// TIA Portal V19 export
FUNCTION "AI SCALING" : Void   // FC5, LAD
{ S7_Optimized_Access := 'TRUE' }
// stored: SetENOAutomatically false
BEGIN

REGION Network 1: OXIDATION REDUCTION POTENTIO METER 301
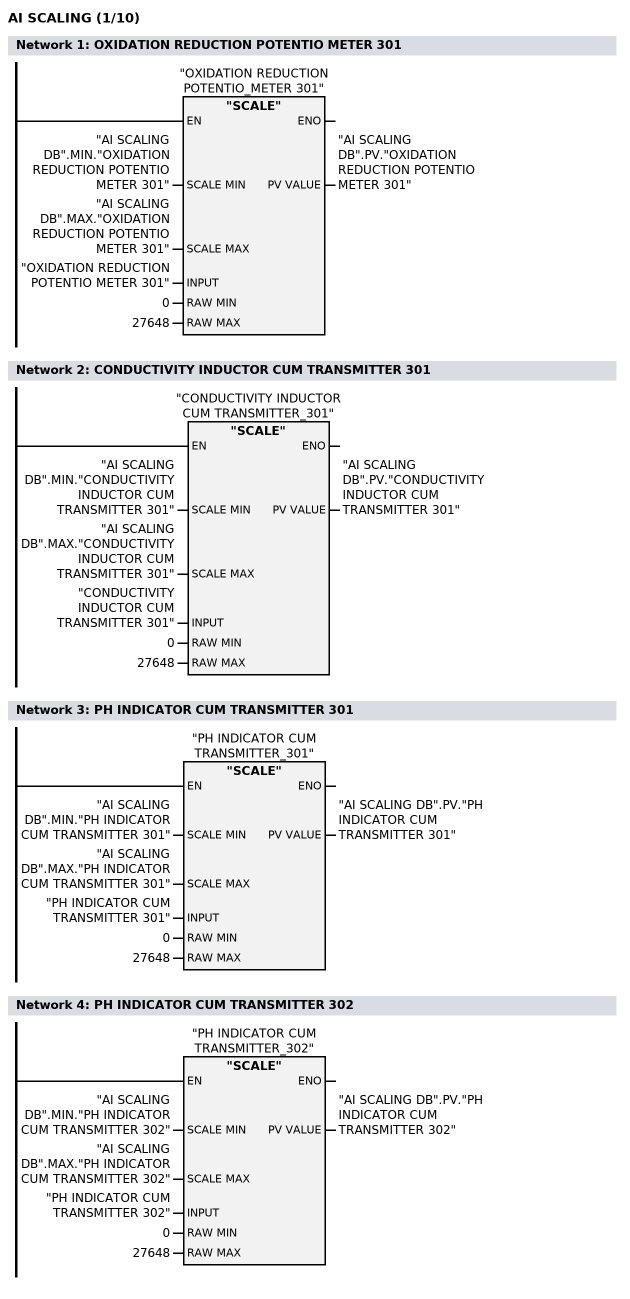
   RUNG wire#powerrail
      "OXIDATION REDUCTION POTENTIO_METER 301"("SCALE MIN" := "AI SCALING DB".MIN."OXIDATION REDUCTION POTENTIO METER 301", "SCALE MAX" := "AI SCALING DB".MAX."OXIDATION REDUCTION POTENTIO METER 301", INPUT := "OXIDATION REDUCTION POTENTIO METER 301", "RAW MIN" := 0, "RAW MAX" := 27648, "PV VALUE" => "AI SCALING DB".PV."OXIDATION REDUCTION POTENTIO METER 301")
   END_RUNG
   // the same network as SCL:
   "OXIDATION REDUCTION POTENTIO_METER 301"("SCALE MIN" := "AI SCALING DB".MIN."OXIDATION REDUCTION POTENTIO METER 301",   // "SCALE"
                           "SCALE MAX" := "AI SCALING DB".MAX."OXIDATION REDUCTION POTENTIO METER 301",
                           INPUT := "OXIDATION REDUCTION POTENTIO METER 301",
                           "RAW MIN" := 0,
                           "RAW MAX" := 27648,
                           "PV VALUE" => "AI SCALING DB".PV."OXIDATION REDUCTION POTENTIO METER 301");
END_REGION

REGION Network 2: CONDUCTIVITY INDUCTOR CUM TRANSMITTER 301
   RUNG wire#powerrail
      "CONDUCTIVITY INDUCTOR CUM TRANSMITTER_301"("SCALE MIN" := "AI SCALING DB".MIN."CONDUCTIVITY INDUCTOR CUM TRANSMITTER 301", "SCALE MAX" := "AI SCALING DB".MAX."CONDUCTIVITY INDUCTOR CUM TRANSMITTER 301", INPUT := "CONDUCTIVITY INDUCTOR CUM TRANSMITTER 301", "RAW MIN" := 0, "RAW MAX" := 27648, "PV VALUE" => "AI SCALING DB".PV."CONDUCTIVITY INDUCTOR CUM TRANSMITTER 301")
   END_RUNG
   // the same network as SCL:
   "CONDUCTIVITY INDUCTOR CUM TRANSMITTER_301"("SCALE MIN" := "AI SCALING DB".MIN."CONDUCTIVITY INDUCTOR CUM TRANSMITTER 301",   // "SCALE"
                           "SCALE MAX" := "AI SCALING DB".MAX."CONDUCTIVITY INDUCTOR CUM TRANSMITTER 301",
                           INPUT := "CONDUCTIVITY INDUCTOR CUM TRANSMITTER 301",
                           "RAW MIN" := 0,
                           "RAW MAX" := 27648,
                           "PV VALUE" => "AI SCALING DB".PV."CONDUCTIVITY INDUCTOR CUM TRANSMITTER 301");
END_REGION

REGION Network 3: PH INDICATOR CUM TRANSMITTER 301
   RUNG wire#powerrail
      "PH INDICATOR CUM TRANSMITTER_301"("SCALE MIN" := "AI SCALING DB".MIN."PH INDICATOR CUM TRANSMITTER 301", "SCALE MAX" := "AI SCALING DB".MAX."PH INDICATOR CUM TRANSMITTER 301", INPUT := "PH INDICATOR CUM TRANSMITTER 301", "RAW MIN" := 0, "RAW MAX" := 27648, "PV VALUE" => "AI SCALING DB".PV."PH INDICATOR CUM TRANSMITTER 301")
   END_RUNG
   // the same network as SCL:
   "PH INDICATOR CUM TRANSMITTER_301"("SCALE MIN" := "AI SCALING DB".MIN."PH INDICATOR CUM TRANSMITTER 301",   // "SCALE"
                           "SCALE MAX" := "AI SCALING DB".MAX."PH INDICATOR CUM TRANSMITTER 301",
                           INPUT := "PH INDICATOR CUM TRANSMITTER 301",
                           "RAW MIN" := 0,
                           "RAW MAX" := 27648,
                           "PV VALUE" => "AI SCALING DB".PV."PH INDICATOR CUM TRANSMITTER 301");
END_REGION

REGION Network 4: PH INDICATOR CUM TRANSMITTER 302
   RUNG wire#powerrail
      "PH INDICATOR CUM TRANSMITTER_302"("SCALE MIN" := "AI SCALING DB".MIN."PH INDICATOR CUM TRANSMITTER 302", "SCALE MAX" := "AI SCALING DB".MAX."PH INDICATOR CUM TRANSMITTER 302", INPUT := "PH INDICATOR CUM TRANSMITTER 302", "RAW MIN" := 0, "RAW MAX" := 27648, "PV VALUE" => "AI SCALING DB".PV."PH INDICATOR CUM TRANSMITTER 302")
   END_RUNG
   // the same network as SCL:
   "PH INDICATOR CUM TRANSMITTER_302"("SCALE MIN" := "AI SCALING DB".MIN."PH INDICATOR CUM TRANSMITTER 302",   // "SCALE"
                           "SCALE MAX" := "AI SCALING DB".MAX."PH INDICATOR CUM TRANSMITTER 302",
                           INPUT := "PH INDICATOR CUM TRANSMITTER 302",
                           "RAW MIN" := 0,
                           "RAW MAX" := 27648,
                           "PV VALUE" => "AI SCALING DB".PV."PH INDICATOR CUM TRANSMITTER 302");
END_REGION

REGION Network 5: CONDUCTIVITY INDICATOR CUM TRANSMITTER 302
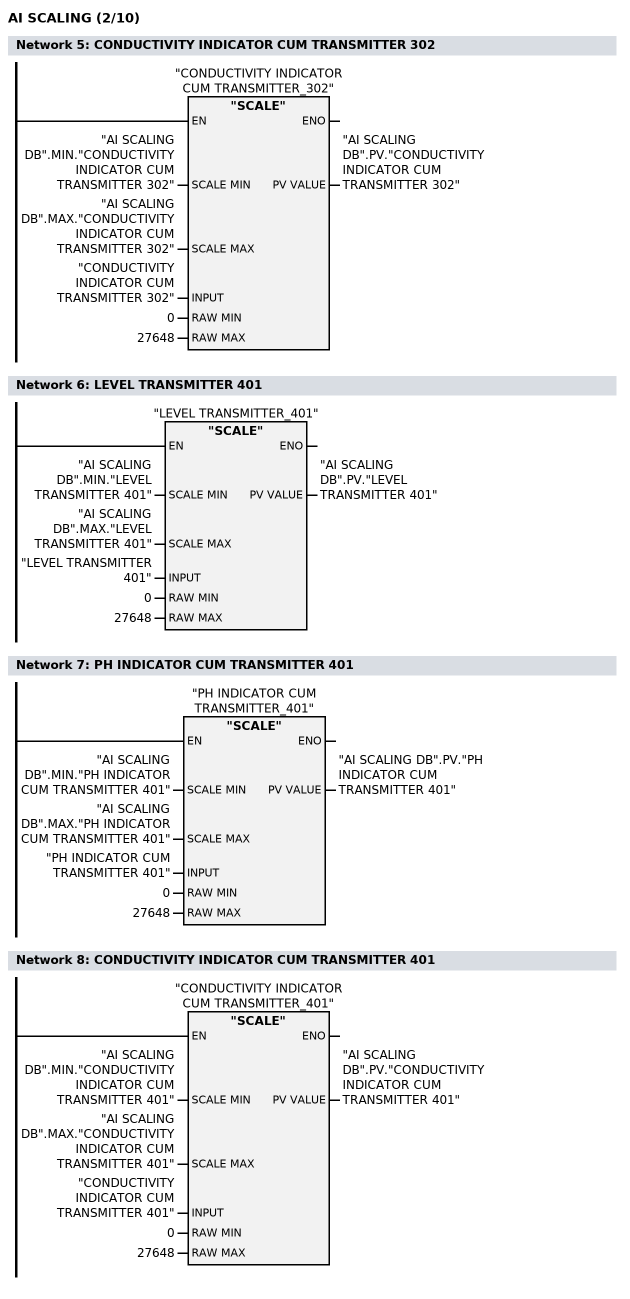
   RUNG wire#powerrail
      "CONDUCTIVITY INDICATOR CUM TRANSMITTER_302"("SCALE MIN" := "AI SCALING DB".MIN."CONDUCTIVITY INDICATOR CUM TRANSMITTER 302", "SCALE MAX" := "AI SCALING DB".MAX."CONDUCTIVITY INDICATOR CUM TRANSMITTER 302", INPUT := "CONDUCTIVITY INDICATOR CUM TRANSMITTER 302", "RAW MIN" := 0, "RAW MAX" := 27648, "PV VALUE" => "AI SCALING DB".PV."CONDUCTIVITY INDICATOR CUM TRANSMITTER 302")
   END_RUNG
   // the same network as SCL:
   "CONDUCTIVITY INDICATOR CUM TRANSMITTER_302"("SCALE MIN" := "AI SCALING DB".MIN."CONDUCTIVITY INDICATOR CUM TRANSMITTER 302",   // "SCALE"
                           "SCALE MAX" := "AI SCALING DB".MAX."CONDUCTIVITY INDICATOR CUM TRANSMITTER 302",
                           INPUT := "CONDUCTIVITY INDICATOR CUM TRANSMITTER 302",
                           "RAW MIN" := 0,
                           "RAW MAX" := 27648,
                           "PV VALUE" => "AI SCALING DB".PV."CONDUCTIVITY INDICATOR CUM TRANSMITTER 302");
END_REGION

REGION Network 6: LEVEL TRANSMITTER 401
   RUNG wire#powerrail
      "LEVEL TRANSMITTER_401"("SCALE MIN" := "AI SCALING DB".MIN."LEVEL TRANSMITTER 401", "SCALE MAX" := "AI SCALING DB".MAX."LEVEL TRANSMITTER 401", INPUT := "LEVEL TRANSMITTER 401", "RAW MIN" := 0, "RAW MAX" := 27648, "PV VALUE" => "AI SCALING DB".PV."LEVEL TRANSMITTER 401")
   END_RUNG
   // the same network as SCL:
   "LEVEL TRANSMITTER_401"("SCALE MIN" := "AI SCALING DB".MIN."LEVEL TRANSMITTER 401",   // "SCALE"
                           "SCALE MAX" := "AI SCALING DB".MAX."LEVEL TRANSMITTER 401",
                           INPUT := "LEVEL TRANSMITTER 401",
                           "RAW MIN" := 0,
                           "RAW MAX" := 27648,
                           "PV VALUE" => "AI SCALING DB".PV."LEVEL TRANSMITTER 401");
END_REGION

REGION Network 7: PH INDICATOR CUM TRANSMITTER 401
   RUNG wire#powerrail
      "PH INDICATOR CUM TRANSMITTER_401"("SCALE MIN" := "AI SCALING DB".MIN."PH INDICATOR CUM TRANSMITTER 401", "SCALE MAX" := "AI SCALING DB".MAX."PH INDICATOR CUM TRANSMITTER 401", INPUT := "PH INDICATOR CUM TRANSMITTER 401", "RAW MIN" := 0, "RAW MAX" := 27648, "PV VALUE" => "AI SCALING DB".PV."PH INDICATOR CUM TRANSMITTER 401")
   END_RUNG
   // the same network as SCL:
   "PH INDICATOR CUM TRANSMITTER_401"("SCALE MIN" := "AI SCALING DB".MIN."PH INDICATOR CUM TRANSMITTER 401",   // "SCALE"
                           "SCALE MAX" := "AI SCALING DB".MAX."PH INDICATOR CUM TRANSMITTER 401",
                           INPUT := "PH INDICATOR CUM TRANSMITTER 401",
                           "RAW MIN" := 0,
                           "RAW MAX" := 27648,
                           "PV VALUE" => "AI SCALING DB".PV."PH INDICATOR CUM TRANSMITTER 401");
END_REGION

REGION Network 8: CONDUCTIVITY INDICATOR CUM TRANSMITTER 401
   RUNG wire#powerrail
      "CONDUCTIVITY INDICATOR CUM TRANSMITTER_401"("SCALE MIN" := "AI SCALING DB".MIN."CONDUCTIVITY INDICATOR CUM TRANSMITTER 401", "SCALE MAX" := "AI SCALING DB".MAX."CONDUCTIVITY INDICATOR CUM TRANSMITTER 401", INPUT := "CONDUCTIVITY INDICATOR CUM TRANSMITTER 401", "RAW MIN" := 0, "RAW MAX" := 27648, "PV VALUE" => "AI SCALING DB".PV."CONDUCTIVITY INDICATOR CUM TRANSMITTER 401")
   END_RUNG
   // the same network as SCL:
   "CONDUCTIVITY INDICATOR CUM TRANSMITTER_401"("SCALE MIN" := "AI SCALING DB".MIN."CONDUCTIVITY INDICATOR CUM TRANSMITTER 401",   // "SCALE"
                           "SCALE MAX" := "AI SCALING DB".MAX."CONDUCTIVITY INDICATOR CUM TRANSMITTER 401",
                           INPUT := "CONDUCTIVITY INDICATOR CUM TRANSMITTER 401",
                           "RAW MIN" := 0,
                           "RAW MAX" := 27648,
                           "PV VALUE" => "AI SCALING DB".PV."CONDUCTIVITY INDICATOR CUM TRANSMITTER 401");
END_REGION

REGION Network 9: CONFUCTIVITY INDICATOR CUM TRANSMITTER 402
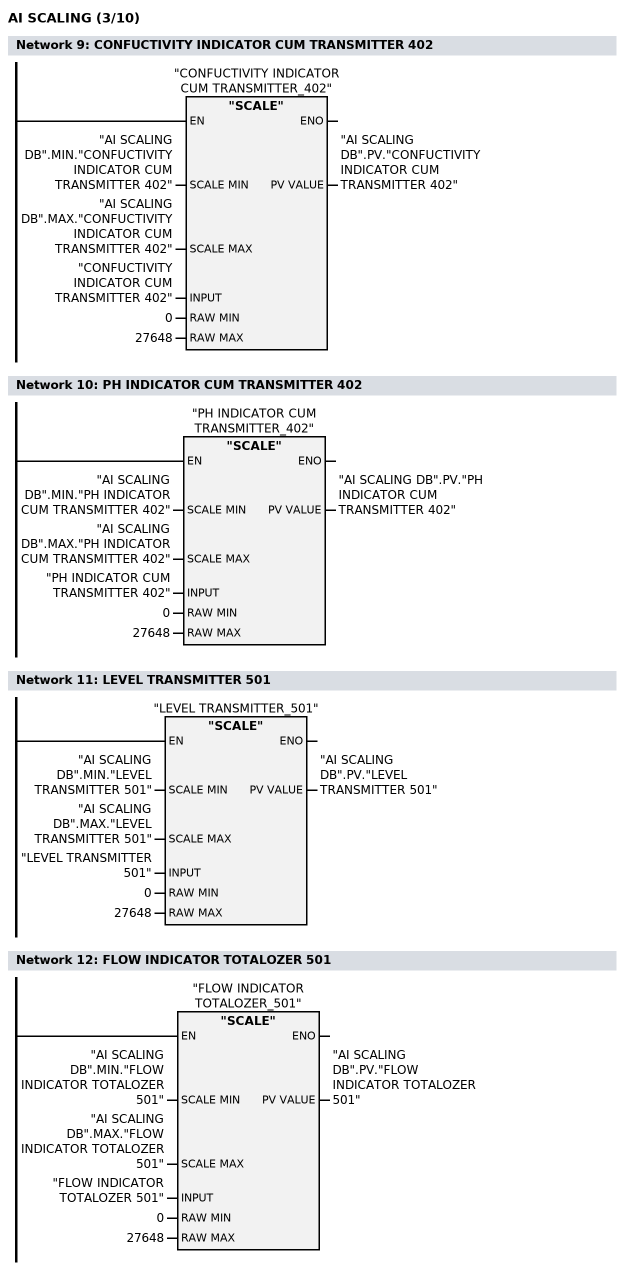
   RUNG wire#powerrail
      "CONFUCTIVITY INDICATOR CUM TRANSMITTER_402"("SCALE MIN" := "AI SCALING DB".MIN."CONFUCTIVITY INDICATOR CUM TRANSMITTER 402", "SCALE MAX" := "AI SCALING DB".MAX."CONFUCTIVITY INDICATOR CUM TRANSMITTER 402", INPUT := "CONFUCTIVITY INDICATOR CUM TRANSMITTER 402", "RAW MIN" := 0, "RAW MAX" := 27648, "PV VALUE" => "AI SCALING DB".PV."CONFUCTIVITY INDICATOR CUM TRANSMITTER 402")
   END_RUNG
   // the same network as SCL:
   "CONFUCTIVITY INDICATOR CUM TRANSMITTER_402"("SCALE MIN" := "AI SCALING DB".MIN."CONFUCTIVITY INDICATOR CUM TRANSMITTER 402",   // "SCALE"
                           "SCALE MAX" := "AI SCALING DB".MAX."CONFUCTIVITY INDICATOR CUM TRANSMITTER 402",
                           INPUT := "CONFUCTIVITY INDICATOR CUM TRANSMITTER 402",
                           "RAW MIN" := 0,
                           "RAW MAX" := 27648,
                           "PV VALUE" => "AI SCALING DB".PV."CONFUCTIVITY INDICATOR CUM TRANSMITTER 402");
END_REGION

REGION Network 10: PH INDICATOR CUM TRANSMITTER 402
   RUNG wire#powerrail
      "PH INDICATOR CUM TRANSMITTER_402"("SCALE MIN" := "AI SCALING DB".MIN."PH INDICATOR CUM TRANSMITTER 402", "SCALE MAX" := "AI SCALING DB".MAX."PH INDICATOR CUM TRANSMITTER 402", INPUT := "PH INDICATOR CUM TRANSMITTER 402", "RAW MIN" := 0, "RAW MAX" := 27648, "PV VALUE" => "AI SCALING DB".PV."PH INDICATOR CUM TRANSMITTER 402")
   END_RUNG
   // the same network as SCL:
   "PH INDICATOR CUM TRANSMITTER_402"("SCALE MIN" := "AI SCALING DB".MIN."PH INDICATOR CUM TRANSMITTER 402",   // "SCALE"
                           "SCALE MAX" := "AI SCALING DB".MAX."PH INDICATOR CUM TRANSMITTER 402",
                           INPUT := "PH INDICATOR CUM TRANSMITTER 402",
                           "RAW MIN" := 0,
                           "RAW MAX" := 27648,
                           "PV VALUE" => "AI SCALING DB".PV."PH INDICATOR CUM TRANSMITTER 402");
END_REGION

REGION Network 11: LEVEL TRANSMITTER 501
   RUNG wire#powerrail
      "LEVEL TRANSMITTER_501"("SCALE MIN" := "AI SCALING DB".MIN."LEVEL TRANSMITTER 501", "SCALE MAX" := "AI SCALING DB".MAX."LEVEL TRANSMITTER 501", INPUT := "LEVEL TRANSMITTER 501", "RAW MIN" := 0, "RAW MAX" := 27648, "PV VALUE" => "AI SCALING DB".PV."LEVEL TRANSMITTER 501")
   END_RUNG
   // the same network as SCL:
   "LEVEL TRANSMITTER_501"("SCALE MIN" := "AI SCALING DB".MIN."LEVEL TRANSMITTER 501",   // "SCALE"
                           "SCALE MAX" := "AI SCALING DB".MAX."LEVEL TRANSMITTER 501",
                           INPUT := "LEVEL TRANSMITTER 501",
                           "RAW MIN" := 0,
                           "RAW MAX" := 27648,
                           "PV VALUE" => "AI SCALING DB".PV."LEVEL TRANSMITTER 501");
END_REGION

REGION Network 12: FLOW INDICATOR TOTALOZER 501
   RUNG wire#powerrail
      "FLOW INDICATOR TOTALOZER_501"("SCALE MIN" := "AI SCALING DB".MIN."FLOW INDICATOR TOTALOZER 501", "SCALE MAX" := "AI SCALING DB".MAX."FLOW INDICATOR TOTALOZER 501", INPUT := "FLOW INDICATOR TOTALOZER 501", "RAW MIN" := 0, "RAW MAX" := 27648, "PV VALUE" => "AI SCALING DB".PV."FLOW INDICATOR TOTALOZER 501")
   END_RUNG
   // the same network as SCL:
   "FLOW INDICATOR TOTALOZER_501"("SCALE MIN" := "AI SCALING DB".MIN."FLOW INDICATOR TOTALOZER 501",   // "SCALE"
                           "SCALE MAX" := "AI SCALING DB".MAX."FLOW INDICATOR TOTALOZER 501",
                           INPUT := "FLOW INDICATOR TOTALOZER 501",
                           "RAW MIN" := 0,
                           "RAW MAX" := 27648,
                           "PV VALUE" => "AI SCALING DB".PV."FLOW INDICATOR TOTALOZER 501");
END_REGION

REGION Network 13: PRESSURE TRANSMITTER 501
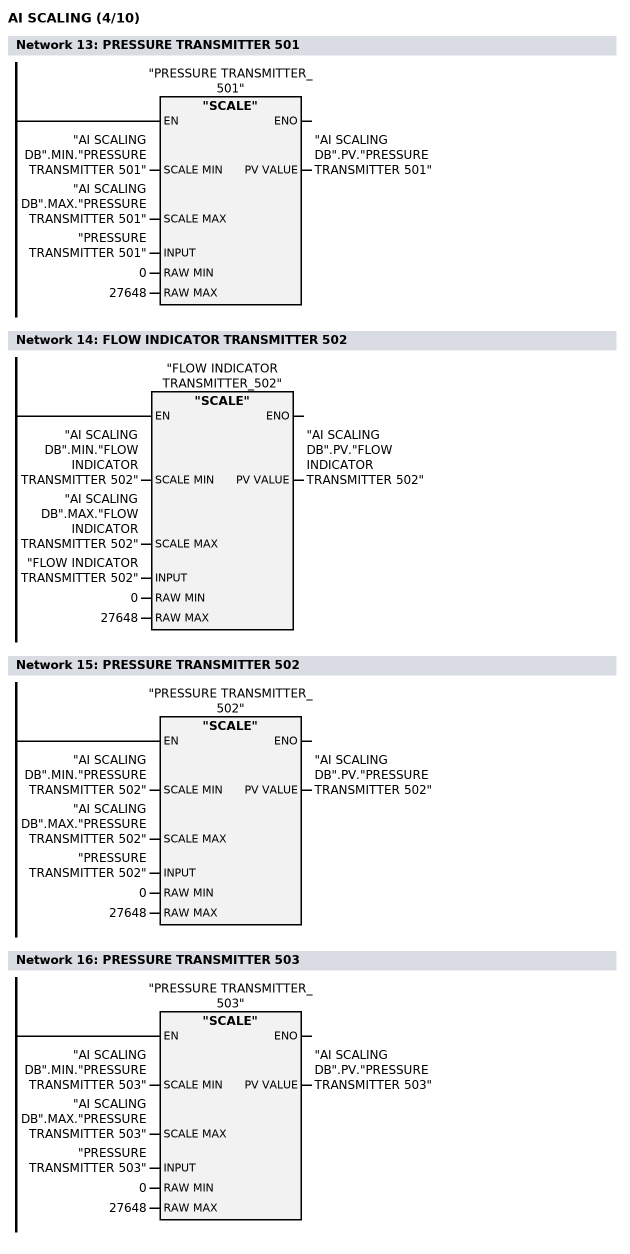
   RUNG wire#powerrail
      "PRESSURE TRANSMITTER_501"("SCALE MIN" := "AI SCALING DB".MIN."PRESSURE TRANSMITTER 501", "SCALE MAX" := "AI SCALING DB".MAX."PRESSURE TRANSMITTER 501", INPUT := "PRESSURE TRANSMITTER 501", "RAW MIN" := 0, "RAW MAX" := 27648, "PV VALUE" => "AI SCALING DB".PV."PRESSURE TRANSMITTER 501")
   END_RUNG
   // the same network as SCL:
   "PRESSURE TRANSMITTER_501"("SCALE MIN" := "AI SCALING DB".MIN."PRESSURE TRANSMITTER 501",   // "SCALE"
                           "SCALE MAX" := "AI SCALING DB".MAX."PRESSURE TRANSMITTER 501",
                           INPUT := "PRESSURE TRANSMITTER 501",
                           "RAW MIN" := 0,
                           "RAW MAX" := 27648,
                           "PV VALUE" => "AI SCALING DB".PV."PRESSURE TRANSMITTER 501");
END_REGION

REGION Network 14: FLOW INDICATOR TRANSMITTER 502
   RUNG wire#powerrail
      "FLOW INDICATOR TRANSMITTER_502"("SCALE MIN" := "AI SCALING DB".MIN."FLOW INDICATOR TRANSMITTER 502", "SCALE MAX" := "AI SCALING DB".MAX."FLOW INDICATOR TRANSMITTER 502", INPUT := "FLOW INDICATOR TRANSMITTER 502", "RAW MIN" := 0, "RAW MAX" := 27648, "PV VALUE" => "AI SCALING DB".PV."FLOW INDICATOR TRANSMITTER 502")
   END_RUNG
   // the same network as SCL:
   "FLOW INDICATOR TRANSMITTER_502"("SCALE MIN" := "AI SCALING DB".MIN."FLOW INDICATOR TRANSMITTER 502",   // "SCALE"
                           "SCALE MAX" := "AI SCALING DB".MAX."FLOW INDICATOR TRANSMITTER 502",
                           INPUT := "FLOW INDICATOR TRANSMITTER 502",
                           "RAW MIN" := 0,
                           "RAW MAX" := 27648,
                           "PV VALUE" => "AI SCALING DB".PV."FLOW INDICATOR TRANSMITTER 502");
END_REGION

REGION Network 15: PRESSURE TRANSMITTER 502
   RUNG wire#powerrail
      "PRESSURE TRANSMITTER_502"("SCALE MIN" := "AI SCALING DB".MIN."PRESSURE TRANSMITTER 502", "SCALE MAX" := "AI SCALING DB".MAX."PRESSURE TRANSMITTER 502", INPUT := "PRESSURE TRANSMITTER 502", "RAW MIN" := 0, "RAW MAX" := 27648, "PV VALUE" => "AI SCALING DB".PV."PRESSURE TRANSMITTER 502")
   END_RUNG
   // the same network as SCL:
   "PRESSURE TRANSMITTER_502"("SCALE MIN" := "AI SCALING DB".MIN."PRESSURE TRANSMITTER 502",   // "SCALE"
                           "SCALE MAX" := "AI SCALING DB".MAX."PRESSURE TRANSMITTER 502",
                           INPUT := "PRESSURE TRANSMITTER 502",
                           "RAW MIN" := 0,
                           "RAW MAX" := 27648,
                           "PV VALUE" => "AI SCALING DB".PV."PRESSURE TRANSMITTER 502");
END_REGION

REGION Network 16: PRESSURE TRANSMITTER 503
   RUNG wire#powerrail
      "PRESSURE TRANSMITTER_503"("SCALE MIN" := "AI SCALING DB".MIN."PRESSURE TRANSMITTER 503", "SCALE MAX" := "AI SCALING DB".MAX."PRESSURE TRANSMITTER 503", INPUT := "PRESSURE TRANSMITTER 503", "RAW MIN" := 0, "RAW MAX" := 27648, "PV VALUE" => "AI SCALING DB".PV."PRESSURE TRANSMITTER 503")
   END_RUNG
   // the same network as SCL:
   "PRESSURE TRANSMITTER_503"("SCALE MIN" := "AI SCALING DB".MIN."PRESSURE TRANSMITTER 503",   // "SCALE"
                           "SCALE MAX" := "AI SCALING DB".MAX."PRESSURE TRANSMITTER 503",
                           INPUT := "PRESSURE TRANSMITTER 503",
                           "RAW MIN" := 0,
                           "RAW MAX" := 27648,
                           "PV VALUE" => "AI SCALING DB".PV."PRESSURE TRANSMITTER 503");
END_REGION

REGION Network 17: PRESSURE TRANSMITTER 504
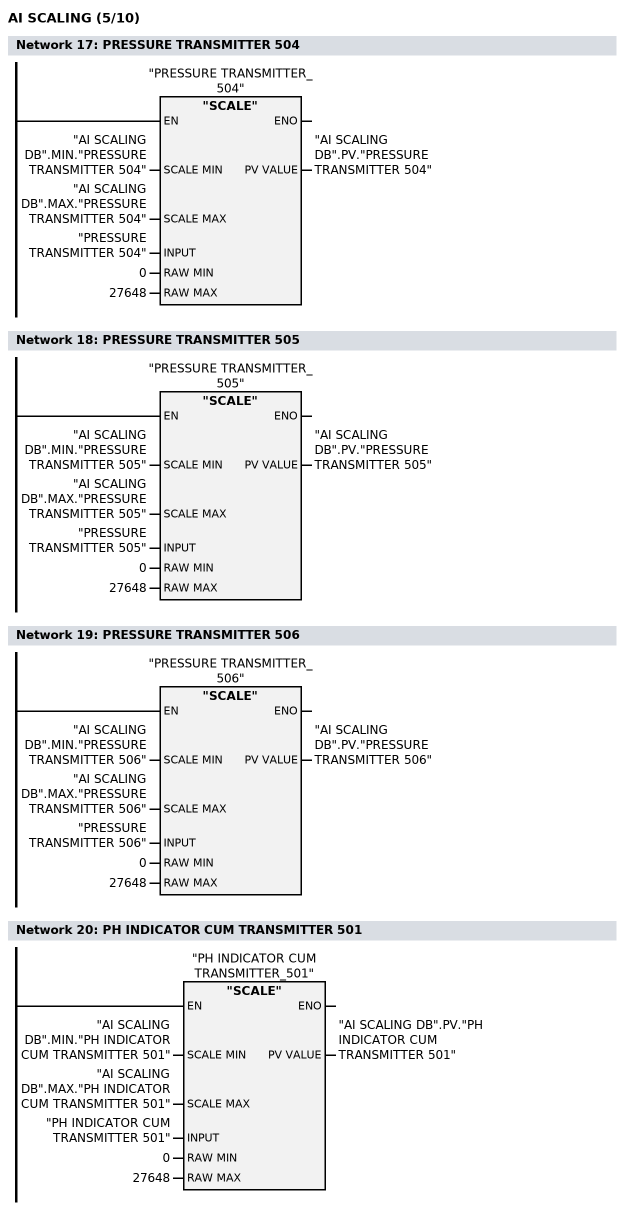
   RUNG wire#powerrail
      "PRESSURE TRANSMITTER_504"("SCALE MIN" := "AI SCALING DB".MIN."PRESSURE TRANSMITTER 504", "SCALE MAX" := "AI SCALING DB".MAX."PRESSURE TRANSMITTER 504", INPUT := "PRESSURE TRANSMITTER 504", "RAW MIN" := 0, "RAW MAX" := 27648, "PV VALUE" => "AI SCALING DB".PV."PRESSURE TRANSMITTER 504")
   END_RUNG
   // the same network as SCL:
   "PRESSURE TRANSMITTER_504"("SCALE MIN" := "AI SCALING DB".MIN."PRESSURE TRANSMITTER 504",   // "SCALE"
                           "SCALE MAX" := "AI SCALING DB".MAX."PRESSURE TRANSMITTER 504",
                           INPUT := "PRESSURE TRANSMITTER 504",
                           "RAW MIN" := 0,
                           "RAW MAX" := 27648,
                           "PV VALUE" => "AI SCALING DB".PV."PRESSURE TRANSMITTER 504");
END_REGION

REGION Network 18: PRESSURE TRANSMITTER 505
   RUNG wire#powerrail
      "PRESSURE TRANSMITTER_505"("SCALE MIN" := "AI SCALING DB".MIN."PRESSURE TRANSMITTER 505", "SCALE MAX" := "AI SCALING DB".MAX."PRESSURE TRANSMITTER 505", INPUT := "PRESSURE TRANSMITTER 505", "RAW MIN" := 0, "RAW MAX" := 27648, "PV VALUE" => "AI SCALING DB".PV."PRESSURE TRANSMITTER 505")
   END_RUNG
   // the same network as SCL:
   "PRESSURE TRANSMITTER_505"("SCALE MIN" := "AI SCALING DB".MIN."PRESSURE TRANSMITTER 505",   // "SCALE"
                           "SCALE MAX" := "AI SCALING DB".MAX."PRESSURE TRANSMITTER 505",
                           INPUT := "PRESSURE TRANSMITTER 505",
                           "RAW MIN" := 0,
                           "RAW MAX" := 27648,
                           "PV VALUE" => "AI SCALING DB".PV."PRESSURE TRANSMITTER 505");
END_REGION

REGION Network 19: PRESSURE TRANSMITTER 506
   RUNG wire#powerrail
      "PRESSURE TRANSMITTER_506"("SCALE MIN" := "AI SCALING DB".MIN."PRESSURE TRANSMITTER 506", "SCALE MAX" := "AI SCALING DB".MAX."PRESSURE TRANSMITTER 506", INPUT := "PRESSURE TRANSMITTER 506", "RAW MIN" := 0, "RAW MAX" := 27648, "PV VALUE" => "AI SCALING DB".PV."PRESSURE TRANSMITTER 506")
   END_RUNG
   // the same network as SCL:
   "PRESSURE TRANSMITTER_506"("SCALE MIN" := "AI SCALING DB".MIN."PRESSURE TRANSMITTER 506",   // "SCALE"
                           "SCALE MAX" := "AI SCALING DB".MAX."PRESSURE TRANSMITTER 506",
                           INPUT := "PRESSURE TRANSMITTER 506",
                           "RAW MIN" := 0,
                           "RAW MAX" := 27648,
                           "PV VALUE" => "AI SCALING DB".PV."PRESSURE TRANSMITTER 506");
END_REGION

REGION Network 20: PH INDICATOR CUM TRANSMITTER 501
   RUNG wire#powerrail
      "PH INDICATOR CUM TRANSMITTER_501"("SCALE MIN" := "AI SCALING DB".MIN."PH INDICATOR CUM TRANSMITTER 501", "SCALE MAX" := "AI SCALING DB".MAX."PH INDICATOR CUM TRANSMITTER 501", INPUT := "PH INDICATOR CUM TRANSMITTER 501", "RAW MIN" := 0, "RAW MAX" := 27648, "PV VALUE" => "AI SCALING DB".PV."PH INDICATOR CUM TRANSMITTER 501")
   END_RUNG
   // the same network as SCL:
   "PH INDICATOR CUM TRANSMITTER_501"("SCALE MIN" := "AI SCALING DB".MIN."PH INDICATOR CUM TRANSMITTER 501",   // "SCALE"
                           "SCALE MAX" := "AI SCALING DB".MAX."PH INDICATOR CUM TRANSMITTER 501",
                           INPUT := "PH INDICATOR CUM TRANSMITTER 501",
                           "RAW MIN" := 0,
                           "RAW MAX" := 27648,
                           "PV VALUE" => "AI SCALING DB".PV."PH INDICATOR CUM TRANSMITTER 501");
END_REGION

REGION Network 21: PH INDICATOR CUM TRANSMITTER 502
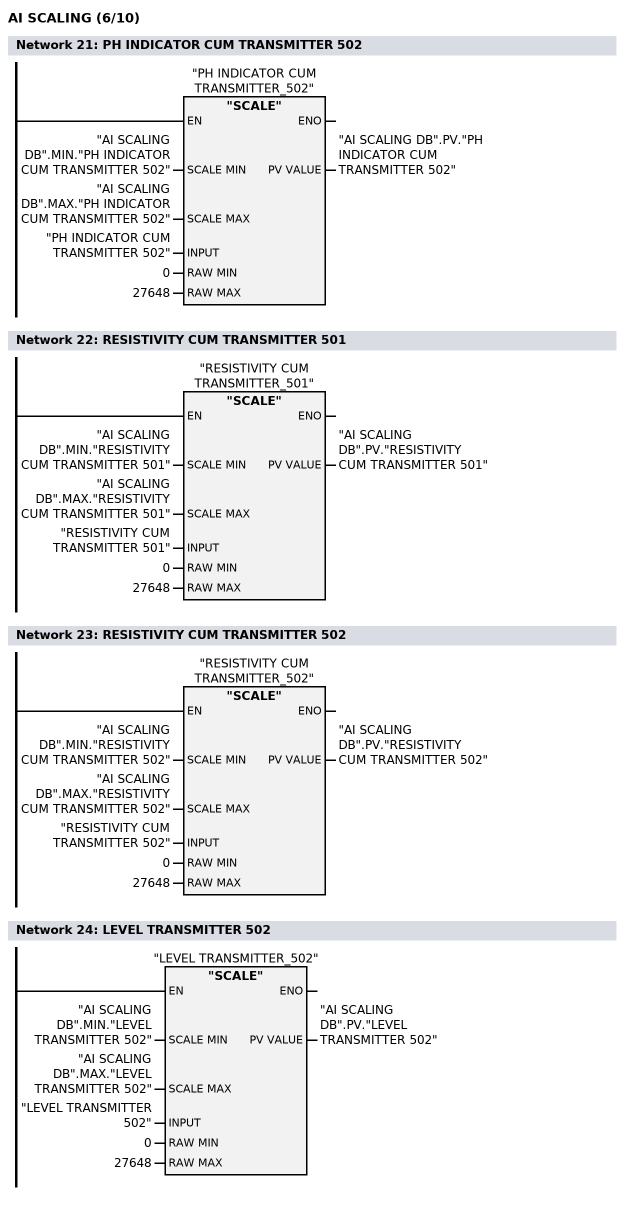
   RUNG wire#powerrail
      "PH INDICATOR CUM TRANSMITTER_502"("SCALE MIN" := "AI SCALING DB".MIN."PH INDICATOR CUM TRANSMITTER 502", "SCALE MAX" := "AI SCALING DB".MAX."PH INDICATOR CUM TRANSMITTER 502", INPUT := "PH INDICATOR CUM TRANSMITTER 502", "RAW MIN" := 0, "RAW MAX" := 27648, "PV VALUE" => "AI SCALING DB".PV."PH INDICATOR CUM TRANSMITTER 502")
   END_RUNG
   // the same network as SCL:
   "PH INDICATOR CUM TRANSMITTER_502"("SCALE MIN" := "AI SCALING DB".MIN."PH INDICATOR CUM TRANSMITTER 502",   // "SCALE"
                           "SCALE MAX" := "AI SCALING DB".MAX."PH INDICATOR CUM TRANSMITTER 502",
                           INPUT := "PH INDICATOR CUM TRANSMITTER 502",
                           "RAW MIN" := 0,
                           "RAW MAX" := 27648,
                           "PV VALUE" => "AI SCALING DB".PV."PH INDICATOR CUM TRANSMITTER 502");
END_REGION

REGION Network 22: RESISTIVITY CUM TRANSMITTER 501
   RUNG wire#powerrail
      "RESISTIVITY CUM TRANSMITTER_501"("SCALE MIN" := "AI SCALING DB".MIN."RESISTIVITY CUM TRANSMITTER 501", "SCALE MAX" := "AI SCALING DB".MAX."RESISTIVITY CUM TRANSMITTER 501", INPUT := "RESISTIVITY CUM TRANSMITTER 501", "RAW MIN" := 0, "RAW MAX" := 27648, "PV VALUE" => "AI SCALING DB".PV."RESISTIVITY CUM TRANSMITTER 501")
   END_RUNG
   // the same network as SCL:
   "RESISTIVITY CUM TRANSMITTER_501"("SCALE MIN" := "AI SCALING DB".MIN."RESISTIVITY CUM TRANSMITTER 501",   // "SCALE"
                           "SCALE MAX" := "AI SCALING DB".MAX."RESISTIVITY CUM TRANSMITTER 501",
                           INPUT := "RESISTIVITY CUM TRANSMITTER 501",
                           "RAW MIN" := 0,
                           "RAW MAX" := 27648,
                           "PV VALUE" => "AI SCALING DB".PV."RESISTIVITY CUM TRANSMITTER 501");
END_REGION

REGION Network 23: RESISTIVITY CUM TRANSMITTER 502
   RUNG wire#powerrail
      "RESISTIVITY CUM TRANSMITTER_502"("SCALE MIN" := "AI SCALING DB".MIN."RESISTIVITY CUM TRANSMITTER 502", "SCALE MAX" := "AI SCALING DB".MAX."RESISTIVITY CUM TRANSMITTER 502", INPUT := "RESISTIVITY CUM TRANSMITTER 502", "RAW MIN" := 0, "RAW MAX" := 27648, "PV VALUE" => "AI SCALING DB".PV."RESISTIVITY CUM TRANSMITTER 502")
   END_RUNG
   // the same network as SCL:
   "RESISTIVITY CUM TRANSMITTER_502"("SCALE MIN" := "AI SCALING DB".MIN."RESISTIVITY CUM TRANSMITTER 502",   // "SCALE"
                           "SCALE MAX" := "AI SCALING DB".MAX."RESISTIVITY CUM TRANSMITTER 502",
                           INPUT := "RESISTIVITY CUM TRANSMITTER 502",
                           "RAW MIN" := 0,
                           "RAW MAX" := 27648,
                           "PV VALUE" => "AI SCALING DB".PV."RESISTIVITY CUM TRANSMITTER 502");
END_REGION

REGION Network 24: LEVEL TRANSMITTER 502
   RUNG wire#powerrail
      "LEVEL TRANSMITTER_502"("SCALE MIN" := "AI SCALING DB".MIN."LEVEL TRANSMITTER 502", "SCALE MAX" := "AI SCALING DB".MAX."LEVEL TRANSMITTER 502", INPUT := "LEVEL TRANSMITTER 502", "RAW MIN" := 0, "RAW MAX" := 27648, "PV VALUE" => "AI SCALING DB".PV."LEVEL TRANSMITTER 502")
   END_RUNG
   // the same network as SCL:
   "LEVEL TRANSMITTER_502"("SCALE MIN" := "AI SCALING DB".MIN."LEVEL TRANSMITTER 502",   // "SCALE"
                           "SCALE MAX" := "AI SCALING DB".MAX."LEVEL TRANSMITTER 502",
                           INPUT := "LEVEL TRANSMITTER 502",
                           "RAW MIN" := 0,
                           "RAW MAX" := 27648,
                           "PV VALUE" => "AI SCALING DB".PV."LEVEL TRANSMITTER 502");
END_REGION

REGION Network 25: FLOW INDICATOR TRANSMITTER 503
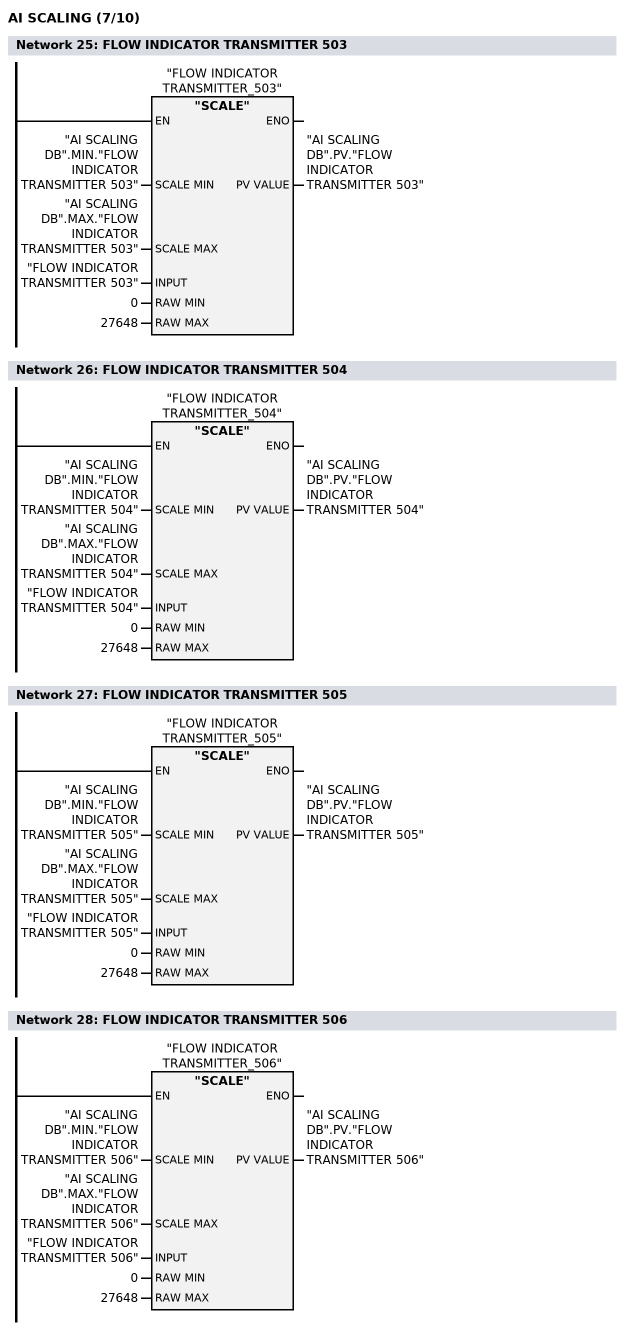
   RUNG wire#powerrail
      "FLOW INDICATOR TRANSMITTER_503"("SCALE MIN" := "AI SCALING DB".MIN."FLOW INDICATOR TRANSMITTER 503", "SCALE MAX" := "AI SCALING DB".MAX."FLOW INDICATOR TRANSMITTER 503", INPUT := "FLOW INDICATOR TRANSMITTER 503", "RAW MIN" := 0, "RAW MAX" := 27648, "PV VALUE" => "AI SCALING DB".PV."FLOW INDICATOR TRANSMITTER 503")
   END_RUNG
   // the same network as SCL:
   "FLOW INDICATOR TRANSMITTER_503"("SCALE MIN" := "AI SCALING DB".MIN."FLOW INDICATOR TRANSMITTER 503",   // "SCALE"
                           "SCALE MAX" := "AI SCALING DB".MAX."FLOW INDICATOR TRANSMITTER 503",
                           INPUT := "FLOW INDICATOR TRANSMITTER 503",
                           "RAW MIN" := 0,
                           "RAW MAX" := 27648,
                           "PV VALUE" => "AI SCALING DB".PV."FLOW INDICATOR TRANSMITTER 503");
END_REGION

REGION Network 26: FLOW INDICATOR TRANSMITTER 504
   RUNG wire#powerrail
      "FLOW INDICATOR TRANSMITTER_504"("SCALE MIN" := "AI SCALING DB".MIN."FLOW INDICATOR TRANSMITTER 504", "SCALE MAX" := "AI SCALING DB".MAX."FLOW INDICATOR TRANSMITTER 504", INPUT := "FLOW INDICATOR TRANSMITTER 504", "RAW MIN" := 0, "RAW MAX" := 27648, "PV VALUE" => "AI SCALING DB".PV."FLOW INDICATOR TRANSMITTER 504")
   END_RUNG
   // the same network as SCL:
   "FLOW INDICATOR TRANSMITTER_504"("SCALE MIN" := "AI SCALING DB".MIN."FLOW INDICATOR TRANSMITTER 504",   // "SCALE"
                           "SCALE MAX" := "AI SCALING DB".MAX."FLOW INDICATOR TRANSMITTER 504",
                           INPUT := "FLOW INDICATOR TRANSMITTER 504",
                           "RAW MIN" := 0,
                           "RAW MAX" := 27648,
                           "PV VALUE" => "AI SCALING DB".PV."FLOW INDICATOR TRANSMITTER 504");
END_REGION

REGION Network 27: FLOW INDICATOR TRANSMITTER 505
   RUNG wire#powerrail
      "FLOW INDICATOR TRANSMITTER_505"("SCALE MIN" := "AI SCALING DB".MIN."FLOW INDICATOR TRANSMITTER 505", "SCALE MAX" := "AI SCALING DB".MAX."FLOW INDICATOR TRANSMITTER 505", INPUT := "FLOW INDICATOR TRANSMITTER 505", "RAW MIN" := 0, "RAW MAX" := 27648, "PV VALUE" => "AI SCALING DB".PV."FLOW INDICATOR TRANSMITTER 505")
   END_RUNG
   // the same network as SCL:
   "FLOW INDICATOR TRANSMITTER_505"("SCALE MIN" := "AI SCALING DB".MIN."FLOW INDICATOR TRANSMITTER 505",   // "SCALE"
                           "SCALE MAX" := "AI SCALING DB".MAX."FLOW INDICATOR TRANSMITTER 505",
                           INPUT := "FLOW INDICATOR TRANSMITTER 505",
                           "RAW MIN" := 0,
                           "RAW MAX" := 27648,
                           "PV VALUE" => "AI SCALING DB".PV."FLOW INDICATOR TRANSMITTER 505");
END_REGION

REGION Network 28: FLOW INDICATOR TRANSMITTER 506
   RUNG wire#powerrail
      "FLOW INDICATOR TRANSMITTER_506"("SCALE MIN" := "AI SCALING DB".MIN."FLOW INDICATOR TRANSMITTER 506", "SCALE MAX" := "AI SCALING DB".MAX."FLOW INDICATOR TRANSMITTER 506", INPUT := "FLOW INDICATOR TRANSMITTER 506", "RAW MIN" := 0, "RAW MAX" := 27648, "PV VALUE" => "AI SCALING DB".PV."FLOW INDICATOR TRANSMITTER 506")
   END_RUNG
   // the same network as SCL:
   "FLOW INDICATOR TRANSMITTER_506"("SCALE MIN" := "AI SCALING DB".MIN."FLOW INDICATOR TRANSMITTER 506",   // "SCALE"
                           "SCALE MAX" := "AI SCALING DB".MAX."FLOW INDICATOR TRANSMITTER 506",
                           INPUT := "FLOW INDICATOR TRANSMITTER 506",
                           "RAW MIN" := 0,
                           "RAW MAX" := 27648,
                           "PV VALUE" => "AI SCALING DB".PV."FLOW INDICATOR TRANSMITTER 506");
END_REGION

REGION Network 29: FLOW INDICATOR TRANSMITTER 507
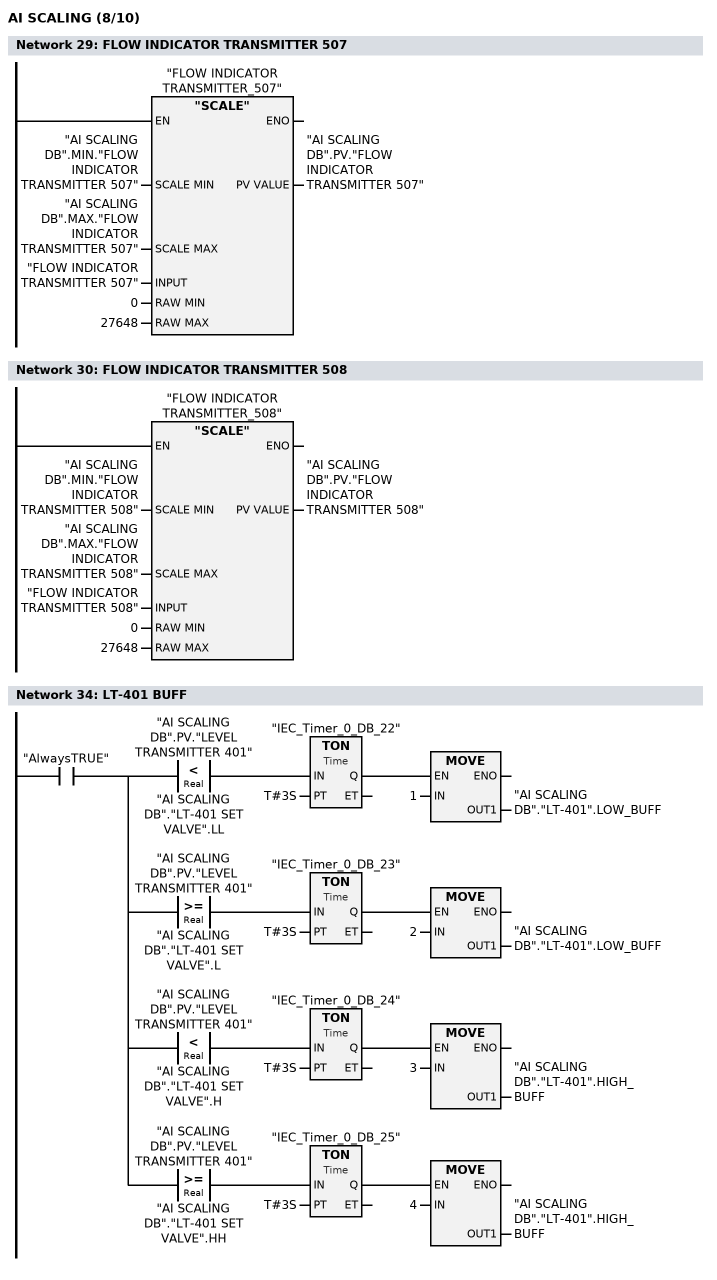
   RUNG wire#powerrail
      "FLOW INDICATOR TRANSMITTER_507"("SCALE MIN" := "AI SCALING DB".MIN."FLOW INDICATOR TRANSMITTER 507", "SCALE MAX" := "AI SCALING DB".MAX."FLOW INDICATOR TRANSMITTER 507", INPUT := "FLOW INDICATOR TRANSMITTER 507", "RAW MIN" := 0, "RAW MAX" := 27648, "PV VALUE" => "AI SCALING DB".PV."FLOW INDICATOR TRANSMITTER 507")
   END_RUNG
   // the same network as SCL:
   "FLOW INDICATOR TRANSMITTER_507"("SCALE MIN" := "AI SCALING DB".MIN."FLOW INDICATOR TRANSMITTER 507",   // "SCALE"
                           "SCALE MAX" := "AI SCALING DB".MAX."FLOW INDICATOR TRANSMITTER 507",
                           INPUT := "FLOW INDICATOR TRANSMITTER 507",
                           "RAW MIN" := 0,
                           "RAW MAX" := 27648,
                           "PV VALUE" => "AI SCALING DB".PV."FLOW INDICATOR TRANSMITTER 507");
END_REGION

REGION Network 30: FLOW INDICATOR TRANSMITTER 508
   RUNG wire#powerrail
      "FLOW INDICATOR TRANSMITTER_508"("SCALE MIN" := "AI SCALING DB".MIN."FLOW INDICATOR TRANSMITTER 508", "SCALE MAX" := "AI SCALING DB".MAX."FLOW INDICATOR TRANSMITTER 508", INPUT := "FLOW INDICATOR TRANSMITTER 508", "RAW MIN" := 0, "RAW MAX" := 27648, "PV VALUE" => "AI SCALING DB".PV."FLOW INDICATOR TRANSMITTER 508")
   END_RUNG
   // the same network as SCL:
   "FLOW INDICATOR TRANSMITTER_508"("SCALE MIN" := "AI SCALING DB".MIN."FLOW INDICATOR TRANSMITTER 508",   // "SCALE"
                           "SCALE MAX" := "AI SCALING DB".MAX."FLOW INDICATOR TRANSMITTER 508",
                           INPUT := "FLOW INDICATOR TRANSMITTER 508",
                           "RAW MIN" := 0,
                           "RAW MAX" := 27648,
                           "PV VALUE" => "AI SCALING DB".PV."FLOW INDICATOR TRANSMITTER 508");
END_REGION

REGION Network 34: LT-401 BUFF
   RUNG wire#powerrail
      Contact( "AlwaysTRUE" )
      wire#w1
      { S7_Templates := "SrcType := Real" } LT_Contact(in1 := "AI SCALING DB".PV."LEVEL TRANSMITTER 401", in2 := "AI SCALING DB"."LT-401 SET VALVE".LL)
      { S7_Templates := "time_type := Time" } "IEC_Timer_0_DB_22".TON(pt := T#3S, et =>)
      Move(in := 1, out1 => "AI SCALING DB"."LT-401".LOW_BUFF)
   END_RUNG
   RUNG wire#w1
      { S7_Templates := "SrcType := Real" } GE_Contact(in1 := "AI SCALING DB".PV."LEVEL TRANSMITTER 401", in2 := "AI SCALING DB"."LT-401 SET VALVE".L)
      { S7_Templates := "time_type := Time" } "IEC_Timer_0_DB_23".TON(pt := T#3S, et =>)
      Move(in := 2, out1 => "AI SCALING DB"."LT-401".LOW_BUFF)
   END_RUNG
   RUNG wire#w1
      { S7_Templates := "SrcType := Real" } LT_Contact(in1 := "AI SCALING DB".PV."LEVEL TRANSMITTER 401", in2 := "AI SCALING DB"."LT-401 SET VALVE".H)
      { S7_Templates := "time_type := Time" } "IEC_Timer_0_DB_24".TON(pt := T#3S, et =>)
      Move(in := 3, out1 => "AI SCALING DB"."LT-401".HIGH_BUFF)
   END_RUNG
   RUNG wire#w1
      { S7_Templates := "SrcType := Real" } GE_Contact(in1 := "AI SCALING DB".PV."LEVEL TRANSMITTER 401", in2 := "AI SCALING DB"."LT-401 SET VALVE".HH)
      { S7_Templates := "time_type := Time" } "IEC_Timer_0_DB_25".TON(pt := T#3S, et =>)
      Move(in := 4, out1 => "AI SCALING DB"."LT-401".HIGH_BUFF)
   END_RUNG
   // the same network as SCL:
   "IEC_Timer_0_DB_22".TON(IN := "AlwaysTRUE" AND ("AI SCALING DB".PV."LEVEL TRANSMITTER 401" < "AI SCALING DB"."LT-401 SET VALVE".LL),
                           PT := T#3S);
   IF "IEC_Timer_0_DB_22".Q THEN "AI SCALING DB"."LT-401".LOW_BUFF := 1; END_IF;
   "IEC_Timer_0_DB_23".TON(IN := "AlwaysTRUE" AND ("AI SCALING DB".PV."LEVEL TRANSMITTER 401" >= "AI SCALING DB"."LT-401 SET VALVE".L),
                           PT := T#3S);
   IF "IEC_Timer_0_DB_23".Q THEN "AI SCALING DB"."LT-401".LOW_BUFF := 2; END_IF;
   "IEC_Timer_0_DB_24".TON(IN := "AlwaysTRUE" AND ("AI SCALING DB".PV."LEVEL TRANSMITTER 401" < "AI SCALING DB"."LT-401 SET VALVE".H),
                           PT := T#3S);
   IF "IEC_Timer_0_DB_24".Q THEN "AI SCALING DB"."LT-401".HIGH_BUFF := 3; END_IF;
   "IEC_Timer_0_DB_25".TON(IN := "AlwaysTRUE" AND ("AI SCALING DB".PV."LEVEL TRANSMITTER 401" >= "AI SCALING DB"."LT-401 SET VALVE".HH),
                           PT := T#3S);
   IF "IEC_Timer_0_DB_25".Q THEN "AI SCALING DB"."LT-401".HIGH_BUFF := 4; END_IF;
END_REGION

REGION Network 35: LT-501 BUFF
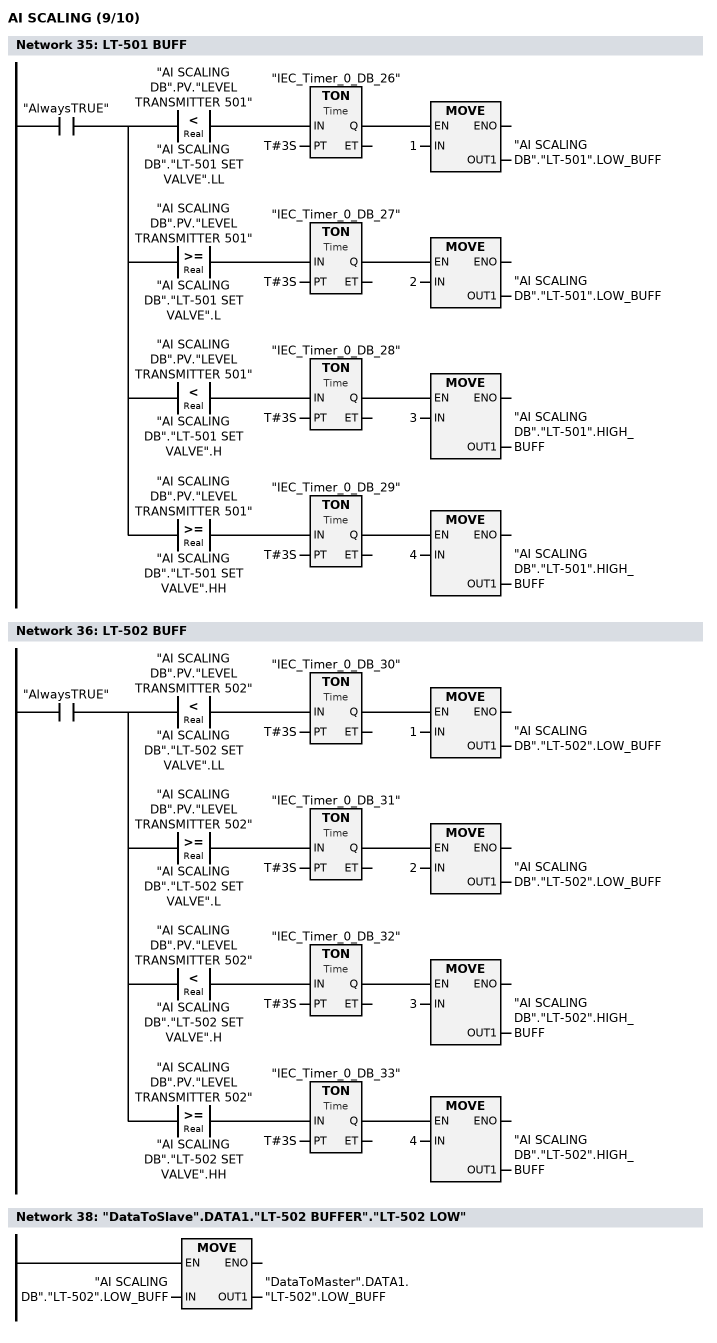
   RUNG wire#powerrail
      Contact( "AlwaysTRUE" )
      wire#w1
      { S7_Templates := "SrcType := Real" } LT_Contact(in1 := "AI SCALING DB".PV."LEVEL TRANSMITTER 501", in2 := "AI SCALING DB"."LT-501 SET VALVE".LL)
      { S7_Templates := "time_type := Time" } "IEC_Timer_0_DB_26".TON(pt := T#3S, et =>)
      Move(in := 1, out1 => "AI SCALING DB"."LT-501".LOW_BUFF)
   END_RUNG
   RUNG wire#w1
      { S7_Templates := "SrcType := Real" } GE_Contact(in1 := "AI SCALING DB".PV."LEVEL TRANSMITTER 501", in2 := "AI SCALING DB"."LT-501 SET VALVE".L)
      { S7_Templates := "time_type := Time" } "IEC_Timer_0_DB_27".TON(pt := T#3S, et =>)
      Move(in := 2, out1 => "AI SCALING DB"."LT-501".LOW_BUFF)
   END_RUNG
   RUNG wire#w1
      { S7_Templates := "SrcType := Real" } LT_Contact(in1 := "AI SCALING DB".PV."LEVEL TRANSMITTER 501", in2 := "AI SCALING DB"."LT-501 SET VALVE".H)
      { S7_Templates := "time_type := Time" } "IEC_Timer_0_DB_28".TON(pt := T#3S, et =>)
      Move(in := 3, out1 => "AI SCALING DB"."LT-501".HIGH_BUFF)
   END_RUNG
   RUNG wire#w1
      { S7_Templates := "SrcType := Real" } GE_Contact(in1 := "AI SCALING DB".PV."LEVEL TRANSMITTER 501", in2 := "AI SCALING DB"."LT-501 SET VALVE".HH)
      { S7_Templates := "time_type := Time" } "IEC_Timer_0_DB_29".TON(pt := T#3S, et =>)
      Move(in := 4, out1 => "AI SCALING DB"."LT-501".HIGH_BUFF)
   END_RUNG
   // the same network as SCL:
   "IEC_Timer_0_DB_26".TON(IN := "AlwaysTRUE" AND ("AI SCALING DB".PV."LEVEL TRANSMITTER 501" < "AI SCALING DB"."LT-501 SET VALVE".LL),
                           PT := T#3S);
   IF "IEC_Timer_0_DB_26".Q THEN "AI SCALING DB"."LT-501".LOW_BUFF := 1; END_IF;
   "IEC_Timer_0_DB_27".TON(IN := "AlwaysTRUE" AND ("AI SCALING DB".PV."LEVEL TRANSMITTER 501" >= "AI SCALING DB"."LT-501 SET VALVE".L),
                           PT := T#3S);
   IF "IEC_Timer_0_DB_27".Q THEN "AI SCALING DB"."LT-501".LOW_BUFF := 2; END_IF;
   "IEC_Timer_0_DB_28".TON(IN := "AlwaysTRUE" AND ("AI SCALING DB".PV."LEVEL TRANSMITTER 501" < "AI SCALING DB"."LT-501 SET VALVE".H),
                           PT := T#3S);
   IF "IEC_Timer_0_DB_28".Q THEN "AI SCALING DB"."LT-501".HIGH_BUFF := 3; END_IF;
   "IEC_Timer_0_DB_29".TON(IN := "AlwaysTRUE" AND ("AI SCALING DB".PV."LEVEL TRANSMITTER 501" >= "AI SCALING DB"."LT-501 SET VALVE".HH),
                           PT := T#3S);
   IF "IEC_Timer_0_DB_29".Q THEN "AI SCALING DB"."LT-501".HIGH_BUFF := 4; END_IF;
END_REGION

REGION Network 36: LT-502 BUFF
   RUNG wire#powerrail
      Contact( "AlwaysTRUE" )
      wire#w1
      { S7_Templates := "SrcType := Real" } LT_Contact(in1 := "AI SCALING DB".PV."LEVEL TRANSMITTER 502", in2 := "AI SCALING DB"."LT-502 SET VALVE".LL)
      { S7_Templates := "time_type := Time" } "IEC_Timer_0_DB_30".TON(pt := T#3S, et =>)
      Move(in := 1, out1 => "AI SCALING DB"."LT-502".LOW_BUFF)
   END_RUNG
   RUNG wire#w1
      { S7_Templates := "SrcType := Real" } GE_Contact(in1 := "AI SCALING DB".PV."LEVEL TRANSMITTER 502", in2 := "AI SCALING DB"."LT-502 SET VALVE".L)
      { S7_Templates := "time_type := Time" } "IEC_Timer_0_DB_31".TON(pt := T#3S, et =>)
      Move(in := 2, out1 => "AI SCALING DB"."LT-502".LOW_BUFF)
   END_RUNG
   RUNG wire#w1
      { S7_Templates := "SrcType := Real" } LT_Contact(in1 := "AI SCALING DB".PV."LEVEL TRANSMITTER 502", in2 := "AI SCALING DB"."LT-502 SET VALVE".H)
      { S7_Templates := "time_type := Time" } "IEC_Timer_0_DB_32".TON(pt := T#3S, et =>)
      Move(in := 3, out1 => "AI SCALING DB"."LT-502".HIGH_BUFF)
   END_RUNG
   RUNG wire#w1
      { S7_Templates := "SrcType := Real" } GE_Contact(in1 := "AI SCALING DB".PV."LEVEL TRANSMITTER 502", in2 := "AI SCALING DB"."LT-502 SET VALVE".HH)
      { S7_Templates := "time_type := Time" } "IEC_Timer_0_DB_33".TON(pt := T#3S, et =>)
      Move(in := 4, out1 => "AI SCALING DB"."LT-502".HIGH_BUFF)
   END_RUNG
   // the same network as SCL:
   "IEC_Timer_0_DB_30".TON(IN := "AlwaysTRUE" AND ("AI SCALING DB".PV."LEVEL TRANSMITTER 502" < "AI SCALING DB"."LT-502 SET VALVE".LL),
                           PT := T#3S);
   IF "IEC_Timer_0_DB_30".Q THEN "AI SCALING DB"."LT-502".LOW_BUFF := 1; END_IF;
   "IEC_Timer_0_DB_31".TON(IN := "AlwaysTRUE" AND ("AI SCALING DB".PV."LEVEL TRANSMITTER 502" >= "AI SCALING DB"."LT-502 SET VALVE".L),
                           PT := T#3S);
   IF "IEC_Timer_0_DB_31".Q THEN "AI SCALING DB"."LT-502".LOW_BUFF := 2; END_IF;
   "IEC_Timer_0_DB_32".TON(IN := "AlwaysTRUE" AND ("AI SCALING DB".PV."LEVEL TRANSMITTER 502" < "AI SCALING DB"."LT-502 SET VALVE".H),
                           PT := T#3S);
   IF "IEC_Timer_0_DB_32".Q THEN "AI SCALING DB"."LT-502".HIGH_BUFF := 3; END_IF;
   "IEC_Timer_0_DB_33".TON(IN := "AlwaysTRUE" AND ("AI SCALING DB".PV."LEVEL TRANSMITTER 502" >= "AI SCALING DB"."LT-502 SET VALVE".HH),
                           PT := T#3S);
   IF "IEC_Timer_0_DB_33".Q THEN "AI SCALING DB"."LT-502".HIGH_BUFF := 4; END_IF;
END_REGION

REGION Network 38: "DataToSlave".DATA1."LT-502 BUFFER"."LT-502 LOW"
   RUNG wire#powerrail
      Move(in := "AI SCALING DB"."LT-502".LOW_BUFF, out1 => "DataToMaster".DATA1."LT-502".LOW_BUFF)
   END_RUNG
   // the same network as SCL:
   "DataToMaster".DATA1."LT-502".LOW_BUFF := "AI SCALING DB"."LT-502".LOW_BUFF;
END_REGION

REGION Network 39: "DataToSlave".DATA1."LT-502 BUFFER"."LT-502 HIGH
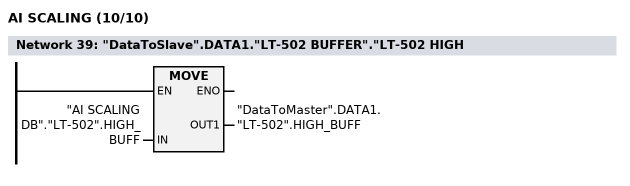
   RUNG wire#powerrail
      Move(in := "AI SCALING DB"."LT-502".HIGH_BUFF, out1 => "DataToMaster".DATA1."LT-502".HIGH_BUFF)
   END_RUNG
   // the same network as SCL:
   "DataToMaster".DATA1."LT-502".HIGH_BUFF := "AI SCALING DB"."LT-502".HIGH_BUFF;
END_REGION
END_FUNCTION
